PROGRAM pouS6Prompts
VAR
	


idbMsgPrompt: FB_CheckMessageBounds;
END_VAR

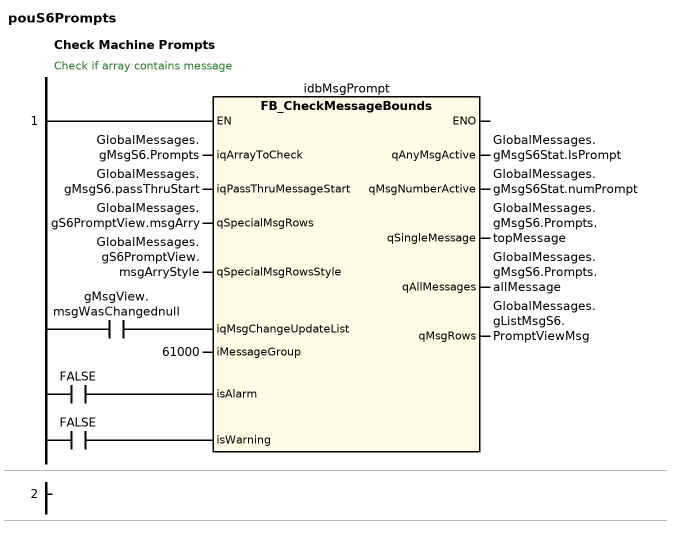
// NETWORK 1: Check Machine Prompts
// Check if array contains message
idbMsgPrompt(
    iqArrayToCheck := GlobalMessages.gMsgS6.Prompts,
    iqPassThruMessageStart := GlobalMessages.gMsgS6.passThruStart,
    qSpecialMsgRows := GlobalMessages.gS6PromptView.msgArry,
    qSpecialMsgRowsStyle := GlobalMessages.gS6PromptView.msgArryStyle,
    iqMsgChangeUpdateList := gMsgView.msgWasChangednull,
    iMessageGroup := 61000,
    isAlarm := FALSE,
    isWarning := FALSE,
    qAnyMsgActive => GlobalMessages.gMsgS6Stat.IsPrompt,
    qMsgNumberActive => GlobalMessages.gMsgS6Stat.numPrompt,
    qSingleMessage => GlobalMessages.gMsgS6.Prompts.topMessage,
    qAllMessages => GlobalMessages.gMsgS6.Prompts.allMessage,
    qMsgRows => GlobalMessages.gListMsgS6.PromptViewMsg); // FB_CheckMessageBounds

// NETWORK 2

END_PROGRAM

(* stored: Version 1.1.0.1, ProductVersion 3.1.4024.11
   POU pouS6Prompts: Id {1b671c62-f677-4124-87af-989471e064aa}, SpecialFunc None *)
